(* CoDeSys 2.3.9.9 project: factory_a.pro *)
(* Libraries: standard.lib 4.10.05 11:14:46, Iecsfc.lib 13.4.06 15:51:28, Util.lib 1.6.07 09:40:58, SysLibTime.lib 18.7.05 09:39:56, SysTaskInfo.lib 18.7.05 09:39:56, SysLibMem.lib 18.7.05 09:39:56, SYSLIBCALLBACK.LIB 18.7.05 09:39:56, BusDiag.LIB 27.8.04 15:06:12, SysExt_AC500_V10.lib 1.7.05 16:17:10, SysInt_AC500_V10.LIB 2.6.06 10:49:48, Ethernet_AC500_V10.LIB 28.7.05 12:19:48 *)

(* PLC configuration (modules and I/O channels)
CPU parameters [AC500_CPU] node 0, in %IB0 out %QB0 {AutoRunType = On; ErrLEDType = On; CheckBatteryType = On; OutputsInStopType = Off in hardware and online; StopErrorClassType = No effect; WarmstartOnFK2Type = Off; FloatingPointExceptionType = E2 failure; IOSimulationModeType = Off; NumberRetainSegmentsType = 8; StartRetainM0Type = 0; EndRetainM0Type = 0; StartRetainM1Type = 0; EndRetainM1Type = 0; StartRetainM2Type = 0; EndRetainM2Type = 0; StartRetainM3Type = 0; EndRetainM3Type = 0; StartRetainM4Type = 0; EndRetainM4Type = 0; StartRetainM5Type = 0; EndRetainM5Type = 0; StartRetainM6Type = 0; EndRetainM6Type = 0; StartRetainM7Type = 0; EndRetainM7Type = 0}
AT %IW0 [WordInputNoSpace] Input 0-15
AT %IB0 [ByteInputNoSpace] Input 0-7
S0 AT %IX0.0 [BoolInput] Input 0
S1 AT %IX0.1 [BoolInput] Input 1
S2 AT %IX0.2 [BoolInput] Input 2
S3 AT %IX0.3 [BoolInput] Input 3
S4 AT %IX0.4 [BoolInput] Input 4
S5 AT %IX0.5 [BoolInput] Input 5
S6 AT %IX0.6 [BoolInput] Input 6
S7 AT %IX0.7 [BoolInput] Input 7
AT %IB1 [ByteInputNoSpace] Input 8-15
S8 AT %IX1.0 [BoolInput] Input 8
S9 AT %IX1.1 [BoolInput] Input 9
S10 AT %IX1.2 [BoolInput] Input 10
S11 AT %IX1.3 [BoolInput] Input 11
S12 AT %IX1.4 [BoolInput] Input 12
S13 AT %IX1.5 [BoolInput] Input 13
S14 AT %IX1.6 [BoolInput] Input 14
S15 AT %IX1.7 [BoolInput] Input 15
AT %IW1 [WordInputNoSpace] Input 16-31
AT %IB2 [ByteInputNoSpace] Input 16-23
AT %IX2.0 [BoolInput] Input 16
AT %IX2.1 [BoolInput] Input 17
AT %IX2.2 [BoolInput] Input 18
AT %IX2.3 [BoolInput] Input 19
AT %IX2.4 [BoolInput] Input 20
AT %IX2.5 [BoolInput] Input 21
AT %IX2.6 [BoolInput] Input 22
AT %IX2.7 [BoolInput] Input 23
AT %IB3 [ByteInputNoSpace] Input 24-31
AT %IX3.0 [BoolInput] Input 24
AT %IX3.1 [BoolInput] Input 25
AT %IX3.2 [BoolInput] Input 26
AT %IX3.3 [BoolInput] Input 27
AT %IX3.4 [BoolInput] Input 28
AT %IX3.5 [BoolInput] Input 29
AT %IX3.6 [BoolInput] Input 30
AT %IX3.7 [BoolInput] Input 31
AT %QW0 [WordOutputNoSpace] Output 16-31
AT %QB0 [ByteOutputNoSpace] Output 16-23
E0 AT %QX0.0 [BoolOutput] Output 16
E1B AT %QX0.1 [BoolOutput] Output 17
E2B AT %QX0.2 [BoolOutput] Output 18
E3 AT %QX0.3 [BoolOutput] Output 19
E4B AT %QX0.4 [BoolOutput] Output 20
E5B AT %QX0.5 [BoolOutput] Output 21
E6B AT %QX0.6 [BoolOutput] Output 22
E7B AT %QX0.7 [BoolOutput] Output 23
AT %QB1 [ByteOutputNoSpace] Output 24-31
AT %QX1.0 [BoolOutput] Output 24
E1F AT %QX1.1 [BoolOutput] Output 25
E2F AT %QX1.2 [BoolOutput] Output 26
AT %QX1.3 [BoolOutput] Output 27
E4F AT %QX1.4 [BoolOutput] Output 28
E5F AT %QX1.5 [BoolOutput] Output 29
E6F AT %QX1.6 [BoolOutput] Output 30
E7F AT %QX1.7 [BoolOutput] Output 31
AT %ID1 [DWordInput] Istwert/Actual value 1
AT %ID2 [DWordInput] Istwert/Actual value 2
AT %IB12 [ByteInputNoBits] Statusbyte/State byte 1
AT %IB13 [ByteInputNoBits] Statusbyte/State byte 2
AT %QD1 [DWordOutput] Startwert/Start value 1
AT %QD2 [DWordOutput] Endwert/End value 1
AT %QD3 [DWordOutput] Startwert/Start value 2
AT %QD4 [DWordOutput] Endwert/End value 2
AT %QB20 [ByteOutputNoBits] Steuerbyte/Control byte 1
AT %QB21 [ByteOutputNoBits] Steuerbyte/Control byte 2
AT %IW7 [WordInputNoSpace] Input 0-15
AT %IB14 [ByteInputNoSpace] Input 0-7
S16 AT %IX14.0 [BoolInput] Input 0
S17 AT %IX14.1 [BoolInput] Input 1
S18 AT %IX14.2 [BoolInput] Input 2
S19 AT %IX14.3 [BoolInput] Input 3
S20 AT %IX14.4 [BoolInput] Input 4
S21 AT %IX14.5 [BoolInput] Input 5
S22 AT %IX14.6 [BoolInput] Input 6
S23 AT %IX14.7 [BoolInput] Input 7
AT %IB15 [ByteInputNoSpace] Input 8-15
S24 AT %IX15.0 [BoolInput] Input 8
S25 AT %IX15.1 [BoolInput] Input 9
S26 AT %IX15.2 [BoolInput] Input 10
S27 AT %IX15.3 [BoolInput] Input 11
AT %IX15.4 [BoolInput] Input 12
AT %IX15.5 [BoolInput] Input 13
AT %IX15.6 [BoolInput] Input 14
SafetyLine_I215 AT %IX15.7 [BoolInput] Input 15
Digital In/Outputs - Inputs 16-31 [Module_16BitInput_16_31] node 1, in %IB16 out %QB22
  AT %IW8 [WordInputNoSpace] Input 16-31
  AT %IB16 [ByteInputNoSpace] Input 16-23
  AT %IX16.0 [BoolInput] Input 16
  AT %IX16.1 [BoolInput] Input 17
  AT %IX16.2 [BoolInput] Input 18
  AT %IX16.3 [BoolInput] Input 19
  AT %IX16.4 [BoolInput] Input 20
  AT %IX16.5 [BoolInput] Input 21
  AT %IX16.6 [BoolInput] Input 22
  AT %IX16.7 [BoolInput] Input 23
  AT %IB17 [ByteInputNoSpace] Input 24-31
  AT %IX17.0 [BoolInput] Input 24
  AT %IX17.1 [BoolInput] Input 25
  AT %IX17.2 [BoolInput] Input 26
  AT %IX17.3 [BoolInput] Input 27
  AT %IX17.4 [BoolInput] Input 28
  AT %IX17.5 [BoolInput] Input 29
  AT %IX17.6 [BoolInput] Input 30
  AT %IX17.7 [BoolInput] Input 31
AT %QW11 [WordOutputNoSpace] Output 16-31
AT %QB22 [ByteOutputNoSpace] Output 16-23
E8B AT %QX22.0 [BoolOutput] Output 16
E9U AT %QX22.1 [BoolOutput] Output 17
AT %QX22.2 [BoolOutput] Output 18
AT %QX22.3 [BoolOutput] Output 19
AT %QX22.4 [BoolOutput] Output 20
AT %QX22.5 [BoolOutput] Output 21
AT %QX22.6 [BoolOutput] Output 22
ALARM AT %QX22.7 [BoolOutput] Output 23
AT %QB23 [ByteOutputNoSpace] Output 24-31
E8F AT %QX23.0 [BoolOutput] Output 24
E9D AT %QX23.1 [BoolOutput] Output 25
AT %QX23.2 [BoolOutput] Output 26
AT %QX23.3 [BoolOutput] Output 27
AT %QX23.4 [BoolOutput] Output 28
AT %QX23.5 [BoolOutput] Output 29
AT %QX23.6 [BoolOutput] Output 30
AT %QX23.7 [BoolOutput] Output 31
AT %ID5 [DWordInput] Istwert/Actual value 1
AT %ID6 [DWordInput] Istwert/Actual value 2
AT %IB28 [ByteInputNoBits] Statusbyte/State byte 1
AT %IB29 [ByteInputNoBits] Statusbyte/State byte 2
AT %QD6 [DWordOutput] Startwert/Start value 1
AT %QD7 [DWordOutput] Endwert/End value 1
AT %QD8 [DWordOutput] Startwert/Start value 2
AT %QD9 [DWordOutput] Endwert/End value 2
AT %QB40 [ByteOutputNoBits] Steuerbyte/Control byte 1
AT %QB41 [ByteOutputNoBits] Steuerbyte/Control byte 2
COM1 - Online access [AC500_COM1_Programming] node 0, in %IB1000 out %QB1000 {COMEnableLoginType = Disabled; COMRTSctrlType = none; COMTLSType = 0; COMCDLYType = 0; COMCharTimeoutType = 0; COMTelEndSelType = none; COMTelEndValCharType = 16#00; COMTelEndValWertType = 0; COMChecksumType = none; COMHandshakeType = none; COMBaudType = 19200; COMParityType = none; COMDataBitType = 8; COMStopBitType = 1}
COM2 - Online access [AC500_COM2_Programming] node 1, in %IB2000 out %QB2000 {COMEnableLoginType = Disabled; COMRTSctrlType = none; COMTLSType = 0; COMCDLYType = 0; COMCharTimeoutType = 0; COMTelEndSelType = none; COMTelEndValCharType = 16#00; COMTelEndValWertType = 0; COMChecksumType = none; COMHandshakeType = none; COMBaudType = 19200; COMParityType = none; COMDataBitType = 8; COMStopBitType = 1}
FBP - none [AC500_FBP_None] node 2, in %IB3000 out %QB3000
MODBUS on TCP/IP [MODBUS_ETH_TCP] node 0, in %IB4000 out %QB4000 {ModbusCouplerOperatingModeType = Master/Slave; COMAdressType = 0; COMDisableWriteStartSeg0Type = 0; COMDisableWriteEndSeg0Type = 0; COMDisableReadStartSeg0Type = 0; COMDisableReadEndSeg0Type = 0; COMDisableWriteStartSeg1Type = 0; COMDisableWriteEndSeg1Type = 0; COMDisableReadStartSeg1Type = 0; COMDisableReadEndSeg1Type = 0}
External - none [AC500_Ext_Empty] node 1, in %IB4000 out %QB4000 {RunConfigFaultType = Yes; MaxWaitRunType = 3000; MinUpdateTimeType = 10; ReserveWord0Type = 0; ReserveWord1Type = 0; ReserveWord2Type = 0}
External - none [AC500_Ext_Empty] node 2, in %IB4000 out %QB4000 {RunConfigFaultType = Yes; MaxWaitRunType = 3000; MinUpdateTimeType = 10; ReserveWord0Type = 0; ReserveWord1Type = 0; ReserveWord2Type = 0}
*)

(* Global variable list: Global_Variables *)
VAR_GLOBAL

	(*Alarms*)
	PressFailureAlarm:BOOL;
	BASE_ALARM:BOOL := FALSE;
	DEFECT_ALARM:BOOL := FALSE;

	(*System variables*)
	AutomaticMode:BOOL :=TRUE;
	Emergency:BOOL :=FALSE;
	SFCInit: BOOL := FALSE;
	SFCReset: BOOL := FALSE;
	EffectorFailureTime: TIME := T#500ms;
	PressStarted:BOOL := FALSE;
	PressFailure:BOOL := FALSE;

	(*Variables for the automatic program*)
	START:BOOL :=FALSE;
	STOP:BOOL :=FALSE;
	RUN:BOOL :=FALSE;
	PRESS_READY:BOOL :=FALSE;
	DIAGNOSTICS_READY:BOOL :=FALSE;
	DEFECT_READY:BOOL :=FALSE;
	ELEVATOR_READY:BOOL :=FALSE;
	LOOK_FOR_PLATES:BOOL :=FALSE;
	NO_BASE_PLATES:BOOL :=FALSE;
	START_PRESS:BOOL :=FALSE;
	LOOK_FOR_BRICKS:BOOL :=FALSE;
	MISSING_BRICKS:BOOL :=FALSE;
	(* Faulty car flag (set by diagnostics) *)
	FAULTY_CAR:BOOL :=FALSE;
	(* Assembly line variables *)
	E0A:BOOL := FALSE;
	E0B:BOOL := FALSE;
	E0C:BOOL := FALSE;
	E0D:BOOL := FALSE;
	E0E:BOOL := FALSE;
	E0F:BOOL := FALSE;
	(* Safe motor variables*)
	E1FS:BOOL := FALSE;
	E1BS:BOOL := FALSE;
	E2FS:BOOL := FALSE;
	E2BS:BOOL := FALSE;
	E3S:BOOL := FALSE;
	E4FS:BOOL := FALSE;
	E4BS:BOOL := FALSE;
	E5FS:BOOL := FALSE;
	E5BS:BOOL := FALSE;
	E6FS:BOOL := FALSE;
	E6BS:BOOL := FALSE;
	E7FS:BOOL := FALSE;
	E7BS:BOOL := FALSE;
	E8FS:BOOL := FALSE;
	E8BS:BOOL := FALSE;
	E9US:BOOL := FALSE;
	E9DS:BOOL := FALSE;
	(* Car detection variables *)
	LOOK_FOR_CAR_PRESS:BOOL :=FALSE;
	CAR_DETECTED_PRESS:BOOL :=FALSE;
	CAR_ARRIVED_PRESS:BOOL :=FALSE;
	LOOK_FOR_CAR_DIAGNOSTICS:BOOL :=FALSE;
	CAR_ARRIVED_DIAGNOSTICS:BOOL :=FALSE;
	LOOK_FOR_CAR_DEFECT:BOOL :=FALSE;
	CAR_DETECTED_DEFECT:BOOL :=FALSE;
	CAR_ARRIVED_DEFECT:BOOL :=FALSE;
	LOOK_FOR_CAR_ELEVATOR:BOOL :=FALSE;
	CAR_DETECTED_ELEVATOR:BOOL :=FALSE;
	CAR_ARRIVED_ELEVATOR:BOOL :=FALSE;
END_VAR

(* POU PLC_PRG, LD *)
PROGRAM PLC_PRG
VAR
	automaticFalling: F_TRIG;
	automaticRising: R_TRIG;
	(* Tachometer *)
	Tacho: BOOL := TRUE;
	TachoTime: TIME := T#240ms;
	TachoTimer1: TON;
	TachoTimer2: TON;
	(* Effector Failure *)
	EffectorFailure: BOOL;
	E1FailureTimer1: TON;
	E1FailureTimer2: TON;
	E1Failure: BOOL;
	E2FailureTimer1: TON;
	E2FailureTimer2: TON;
	E2Failure: BOOL;
	E3FailureTimer: TON;
	E3Failure: BOOL;
	E4FailureTimer1: TON;
	E4FailureTimer2: TON;
	E4Failure: BOOL;
	E5FailureTimer1: TON;
	E5FailureTimer2: TON;
	E5Failure: BOOL;
	E6FailureTimer1: TON;
	E6FailureTimer2: TON;
	E6Failure: BOOL;
	E7FailureTimer1: TON;
	E7FailureTimer2: TON;
	E7Failure: BOOL;
	E8FailureTimer1: TON;
	E8FailureTimer2: TON;
	E8Failure: BOOL;
	E9FailureTimer1: TON;
	E9FailureTimer2: TON;
	E9Failure: BOOL;

	(*Safty press timer, The max press time when press is stuck*)
	(* MaxPressTime:TIME := T#700ms;

	SafetyPressTimer2: TON;
	SafetyPressTimer1: TON;
	Output1: BOOL; *)
END_VAR
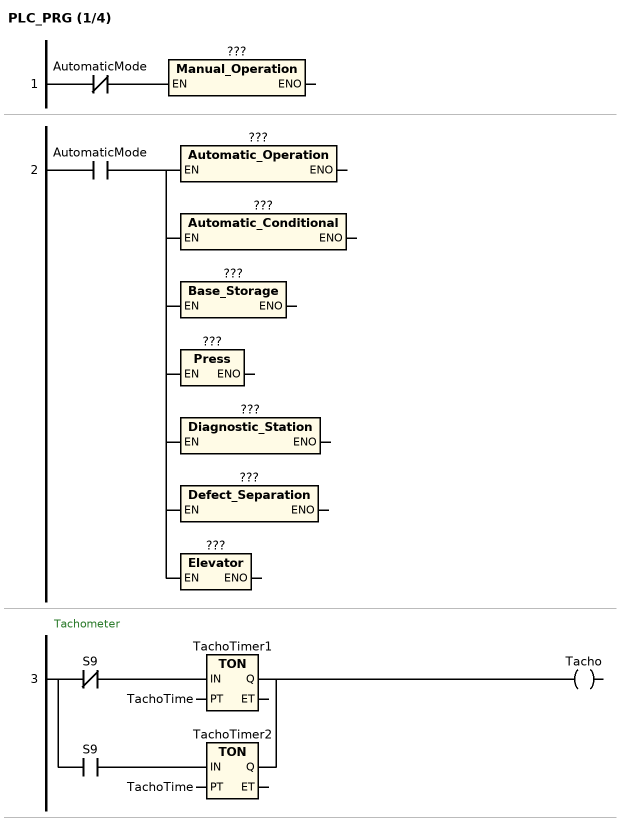
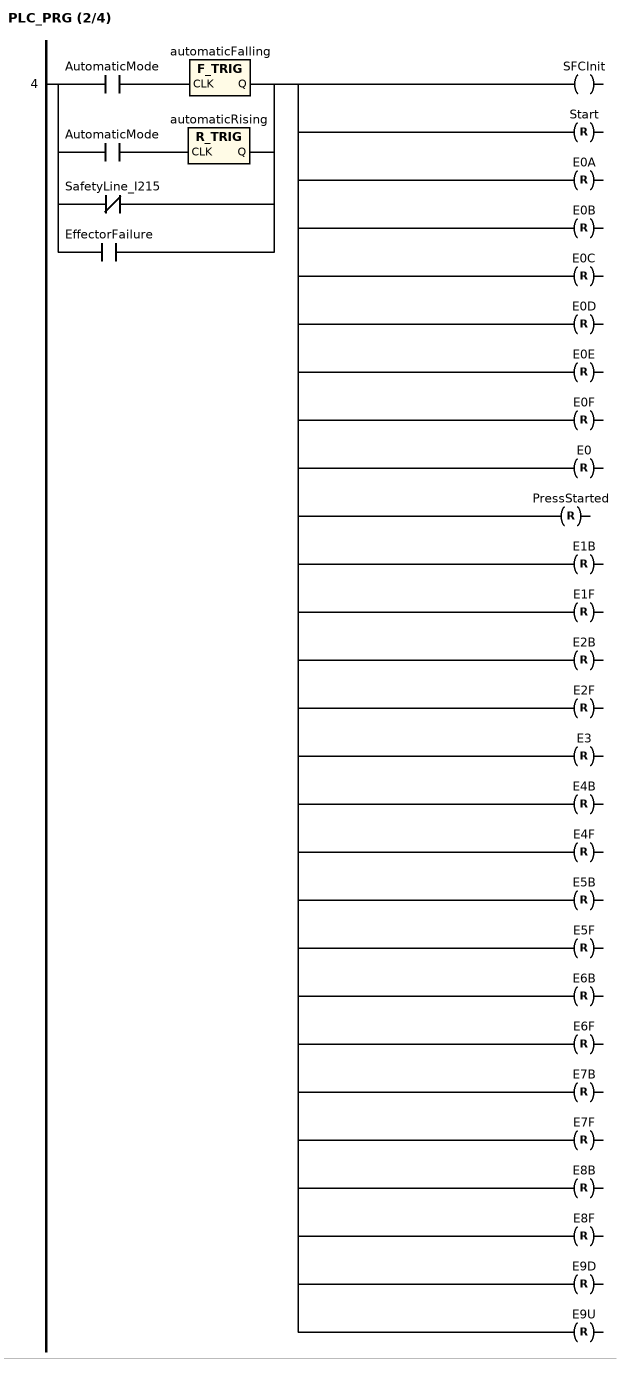
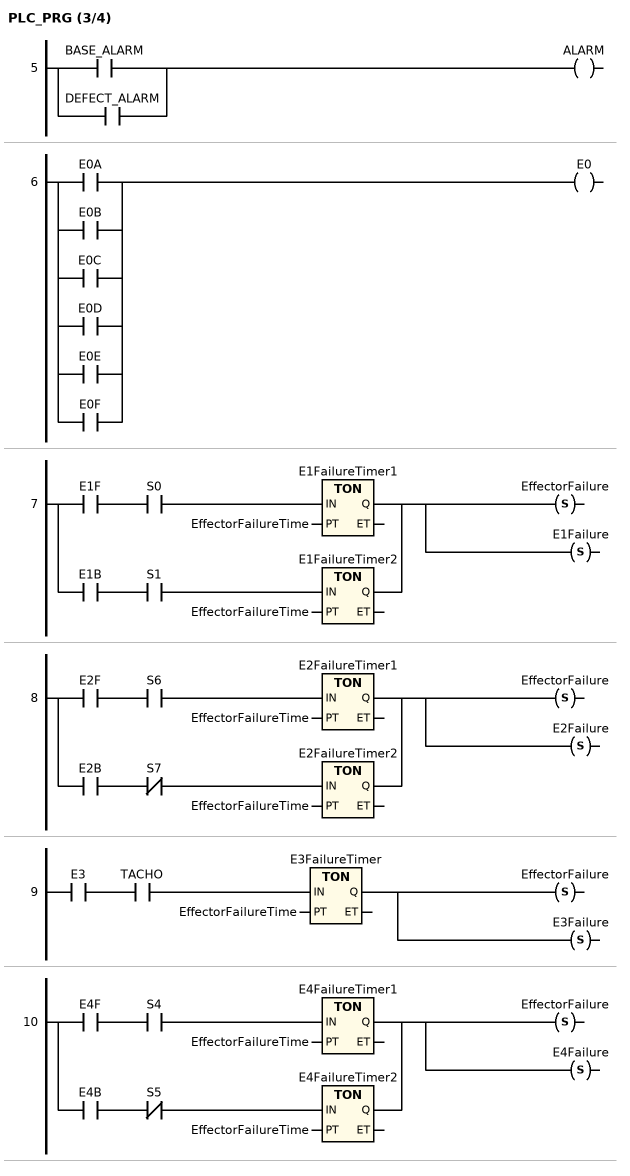
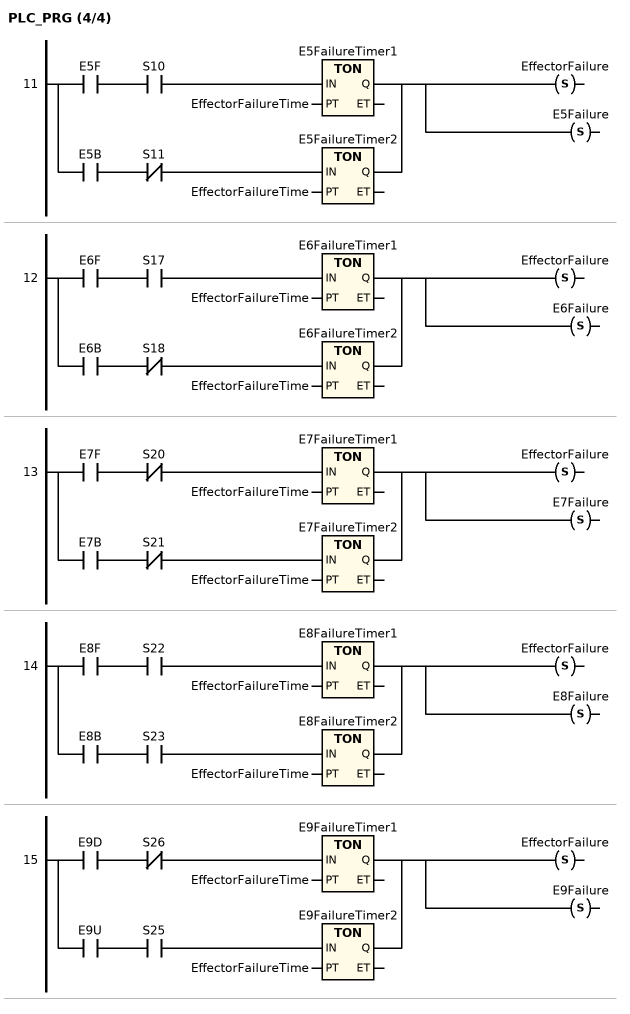
_LD_ (* Ladder Diagram *)
NETWORK 1
	[/AutomaticMode]
		EN --- ???:Manual_Operation()
NETWORK 2
	[AutomaticMode]
		EN --- ???:Automatic_Operation()
		EN --- ???:Automatic_Conditional()
		EN --- ???:Base_Storage()
		EN --- ???:Press()
		EN --- ???:Diagnostic_Station()
		EN --- ???:Defect_Separation()
		EN --- ???:Elevator()
NETWORK 3 (* Tachometer *)
	{ [/S9] - TachoTimer1:TON(IN: *, PT: TachoTime) | [S9] - TachoTimer2:TON(IN: *, PT: TachoTime) } --- (Tacho)
NETWORK 4
	{ [AutomaticMode] - automaticFalling:F_TRIG(CLK: *) | [AutomaticMode] - automaticRising:R_TRIG(CLK: *) | [/SafetyLine_I215] | [EffectorFailure] } --- (SFCInit) (R Start) (R E0A) (R E0B) (R E0C) (R E0D) (R E0E) (R E0F) (R E0) (R PressStarted) (R E1B) (R E1F) (R E2B) (R E2F) (R E3) (R E4B) (R E4F) (R E5B) (R E5F) (R E6B) (R E6F) (R E7B) (R E7F) (R E8B) (R E8F) (R E9D) (R E9U)
NETWORK 5
	{ [BASE_ALARM] | [DEFECT_ALARM] } --- (ALARM)
NETWORK 6
	{ [E0A] | [E0B] | [E0C] | [E0D] | [E0E] | [E0F] } --- (E0)
NETWORK 7
	{ [E1F] - [S0] - E1FailureTimer1:TON(IN: *, PT: EffectorFailureTime) | [E1B] - [S1] - E1FailureTimer2:TON(IN: *, PT: EffectorFailureTime) } --- (S EffectorFailure) (S E1Failure)
NETWORK 8
	{ [E2F] - [S6] - E2FailureTimer1:TON(IN: *, PT: EffectorFailureTime) | [E2B] - [/S7] - E2FailureTimer2:TON(IN: *, PT: EffectorFailureTime) } --- (S EffectorFailure) (S E2Failure)
NETWORK 9
	[E3] - [TACHO] - E3FailureTimer:TON(IN: *, PT: EffectorFailureTime) --- (S EffectorFailure) (S E3Failure)
NETWORK 10
	{ [E4F] - [S4] - E4FailureTimer1:TON(IN: *, PT: EffectorFailureTime) | [E4B] - [/S5] - E4FailureTimer2:TON(IN: *, PT: EffectorFailureTime) } --- (S EffectorFailure) (S E4Failure)
NETWORK 11
	{ [E5F] - [S10] - E5FailureTimer1:TON(IN: *, PT: EffectorFailureTime) | [E5B] - [/S11] - E5FailureTimer2:TON(IN: *, PT: EffectorFailureTime) } --- (S EffectorFailure) (S E5Failure)
NETWORK 12
	{ [E6F] - [S17] - E6FailureTimer1:TON(IN: *, PT: EffectorFailureTime) | [E6B] - [/S18] - E6FailureTimer2:TON(IN: *, PT: EffectorFailureTime) } --- (S EffectorFailure) (S E6Failure)
NETWORK 13
	{ [E7F] - [/S20] - E7FailureTimer1:TON(IN: *, PT: EffectorFailureTime) | [E7B] - [/S21] - E7FailureTimer2:TON(IN: *, PT: EffectorFailureTime) } --- (S EffectorFailure) (S E7Failure)
NETWORK 14
	{ [E8F] - [S22] - E8FailureTimer1:TON(IN: *, PT: EffectorFailureTime) | [E8B] - [S23] - E8FailureTimer2:TON(IN: *, PT: EffectorFailureTime) } --- (S EffectorFailure) (S E8Failure)
NETWORK 15
	{ [E9D] - [/S26] - E9FailureTimer1:TON(IN: *, PT: EffectorFailureTime) | [E9U] - [S25] - E9FailureTimer2:TON(IN: *, PT: EffectorFailureTime) } --- (S EffectorFailure) (S E9Failure)
_END_LD_
(* the same logic as Structured Text *)
(* Network 1: see the listing above *)
(* Network 2: see the listing above *)
(* Network 3 *)
TachoTimer1(IN := NOT S9, PT := TachoTime);
TachoTimer2(IN := S9, PT := TachoTime);
Tacho := TachoTimer1.Q OR TachoTimer2.Q;
(* Network 4 *)
automaticFalling(CLK := AutomaticMode);
automaticRising(CLK := AutomaticMode);
SFCInit := automaticFalling.Q OR automaticRising.Q OR NOT SafetyLine_I215 OR EffectorFailure;
IF SFCInit THEN Start := FALSE; E0A := FALSE; E0B := FALSE; E0C := FALSE; E0D := FALSE; E0E := FALSE; E0F := FALSE; E0 := FALSE; PressStarted := FALSE; E1B := FALSE; E1F := FALSE; E2B := FALSE; E2F := FALSE; E3 := FALSE; E4B := FALSE; E4F := FALSE; E5B := FALSE; E5F := FALSE; E6B := FALSE; E6F := FALSE; E7B := FALSE; E7F := FALSE; E8B := FALSE; E8F := FALSE; E9D := FALSE; E9U := FALSE; END_IF;
(* Network 5 *)
ALARM := BASE_ALARM OR DEFECT_ALARM;
(* Network 6 *)
E0 := E0A OR E0B OR E0C OR E0D OR E0E OR E0F;
(* Network 7 *)
E1FailureTimer1(IN := E1F AND S0, PT := EffectorFailureTime);
E1FailureTimer2(IN := E1B AND S1, PT := EffectorFailureTime);
IF E1FailureTimer1.Q OR E1FailureTimer2.Q THEN EffectorFailure := TRUE; E1Failure := TRUE; END_IF;
(* Network 8 *)
E2FailureTimer1(IN := E2F AND S6, PT := EffectorFailureTime);
E2FailureTimer2(IN := E2B AND NOT S7, PT := EffectorFailureTime);
IF E2FailureTimer1.Q OR E2FailureTimer2.Q THEN EffectorFailure := TRUE; E2Failure := TRUE; END_IF;
(* Network 9 *)
E3FailureTimer(IN := E3 AND TACHO, PT := EffectorFailureTime);
IF E3FailureTimer.Q THEN EffectorFailure := TRUE; E3Failure := TRUE; END_IF;
(* Network 10 *)
E4FailureTimer1(IN := E4F AND S4, PT := EffectorFailureTime);
E4FailureTimer2(IN := E4B AND NOT S5, PT := EffectorFailureTime);
IF E4FailureTimer1.Q OR E4FailureTimer2.Q THEN EffectorFailure := TRUE; E4Failure := TRUE; END_IF;
(* Network 11 *)
E5FailureTimer1(IN := E5F AND S10, PT := EffectorFailureTime);
E5FailureTimer2(IN := E5B AND NOT S11, PT := EffectorFailureTime);
IF E5FailureTimer1.Q OR E5FailureTimer2.Q THEN EffectorFailure := TRUE; E5Failure := TRUE; END_IF;
(* Network 12 *)
E6FailureTimer1(IN := E6F AND S17, PT := EffectorFailureTime);
E6FailureTimer2(IN := E6B AND NOT S18, PT := EffectorFailureTime);
IF E6FailureTimer1.Q OR E6FailureTimer2.Q THEN EffectorFailure := TRUE; E6Failure := TRUE; END_IF;
(* Network 13 *)
E7FailureTimer1(IN := E7F AND NOT S20, PT := EffectorFailureTime);
E7FailureTimer2(IN := E7B AND NOT S21, PT := EffectorFailureTime);
IF E7FailureTimer1.Q OR E7FailureTimer2.Q THEN EffectorFailure := TRUE; E7Failure := TRUE; END_IF;
(* Network 14 *)
E8FailureTimer1(IN := E8F AND S22, PT := EffectorFailureTime);
E8FailureTimer2(IN := E8B AND S23, PT := EffectorFailureTime);
IF E8FailureTimer1.Q OR E8FailureTimer2.Q THEN EffectorFailure := TRUE; E8Failure := TRUE; END_IF;
(* Network 15 *)
E9FailureTimer1(IN := E9D AND NOT S26, PT := EffectorFailureTime);
E9FailureTimer2(IN := E9U AND S25, PT := EffectorFailureTime);
IF E9FailureTimer1.Q OR E9FailureTimer2.Q THEN EffectorFailure := TRUE; E9Failure := TRUE; END_IF;
END_PROGRAM

(* POU Manual_Operation, SFC *)
PROGRAM Manual_Operation
VAR
	StorageAlarmTime:TIME :=T#2S;
	(*E0: Assembly line*)
	(*Not in SFC.Using  E0A directly*)
	(*E1: Base pusher*)
	buttonE1Fwd: BOOL := FALSE;
	buttonE1Bwd: BOOL := FALSE;
	(*E2: Undercarriage pusher*)
	buttonE2Fwd: BOOL := FALSE;
	buttonE2Bwd: BOOL := FALSE;
	(*E3: Press
	Observe! that S8 is active low*)
	buttonE3Press: BOOL := FALSE;
	(*E4: Press pusher*)
	buttonE4Fwd: BOOL := FALSE;
	buttonE4Bwd: BOOL := FALSE;
	(*E5: Press bar*)
	buttonE5Fwd: BOOL := FALSE;
	buttonE5Bwd: BOOL := FALSE;
	(*E6: Diagnostic bar
	Observe! that InEngine6 has NOT inverted contact*)
	buttonE6Fwd: BOOL := FALSE;
	buttonE6Bwd: BOOL := FALSE;
	(*E7: Defect pusher*)
	TimeOutStorage: BOOL := FALSE;
	buttonE7Fwd: BOOL := FALSE;
	buttonE7Bwd: BOOL := FALSE;
	(*E8: Defect bar*)
	buttonE8Fwd: BOOL := FALSE;
	buttonE8Bwd: BOOL := FALSE;
	(*E9: Elevator*)
	buttonE9Up: BOOL := FALSE;
	buttonE9Down: BOOL := FALSE;
END_VAR
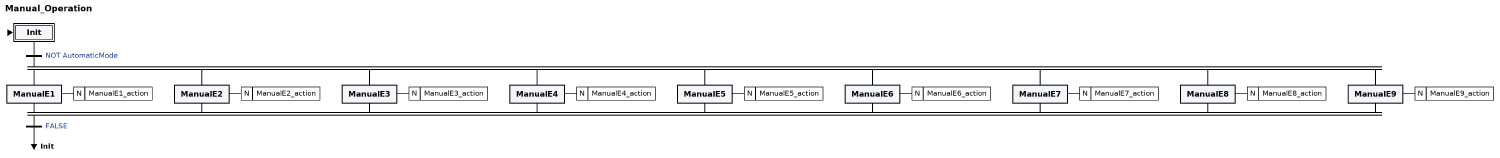
INITIAL_STEP Init:
END_STEP
TRANSITION FROM Init TO (ManualE1, ManualE2, ManualE3, ManualE4, ManualE5, ManualE6, ManualE7, ManualE8, ManualE9) := NOT AutomaticMode;
END_TRANSITION
STEP ManualE1:
	ManualE1_action(N);
END_STEP
STEP ManualE2:
	ManualE2_action(N);
END_STEP
STEP ManualE3:
	ManualE3_action(N);
END_STEP
STEP ManualE4:
	ManualE4_action(N);
END_STEP
STEP ManualE5:
	ManualE5_action(N);
END_STEP
STEP ManualE6:
	ManualE6_action(N);
END_STEP
STEP ManualE7:
	ManualE7_action(N);
END_STEP
STEP ManualE8:
	ManualE8_action(N);
END_STEP
STEP ManualE9:
	ManualE9_action(N);
END_STEP
TRANSITION FROM (ManualE1, ManualE2, ManualE3, ManualE4, ManualE5, ManualE6, ManualE7, ManualE8, ManualE9) TO Init := FALSE;
END_TRANSITION

ACTION ManualE1_action:
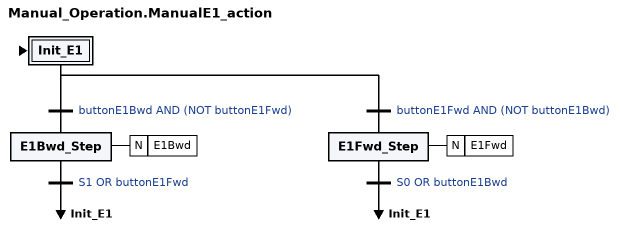
INITIAL_STEP Init_E1:
END_STEP
TRANSITION FROM Init_E1 TO E1Bwd_Step := buttonE1Bwd AND (NOT buttonE1Fwd);
END_TRANSITION
TRANSITION FROM Init_E1 TO E1Fwd_Step := buttonE1Fwd AND (NOT buttonE1Bwd);
END_TRANSITION
STEP E1Bwd_Step:
	E1Bwd(N);
END_STEP
TRANSITION FROM E1Bwd_Step TO Init_E1 := S1 OR buttonE1Fwd;
END_TRANSITION
STEP E1Fwd_Step:
	E1Fwd(N);
END_STEP
TRANSITION FROM E1Fwd_Step TO Init_E1 := S0 OR buttonE1Bwd;
END_TRANSITION
END_ACTION

ACTION ManualE2_action:
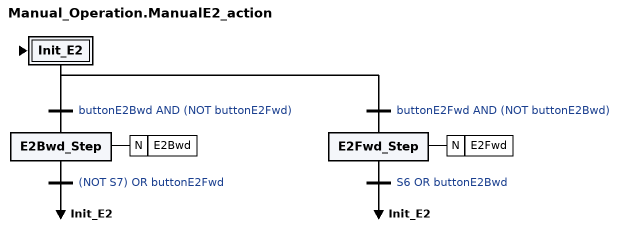
INITIAL_STEP Init_E2:
END_STEP
TRANSITION FROM Init_E2 TO E2Bwd_Step := buttonE2Bwd AND (NOT buttonE2Fwd);
END_TRANSITION
TRANSITION FROM Init_E2 TO E2Fwd_Step := buttonE2Fwd AND (NOT buttonE2Bwd);
END_TRANSITION
STEP E2Bwd_Step:
	E2Bwd(N);
END_STEP
TRANSITION FROM E2Bwd_Step TO Init_E2 := (NOT S7) OR buttonE2Fwd;
END_TRANSITION
STEP E2Fwd_Step:
	E2Fwd(N);
END_STEP
TRANSITION FROM E2Fwd_Step TO Init_E2 := S6 OR buttonE2Bwd;
END_TRANSITION
END_ACTION

ACTION ManualE3_action:
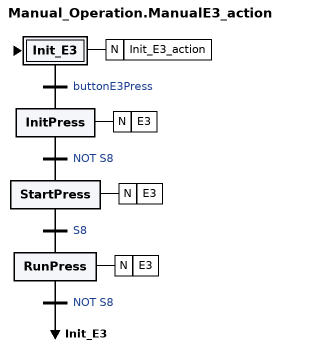
INITIAL_STEP Init_E3:
	Init_E3_action(N);
END_STEP
TRANSITION FROM Init_E3 TO InitPress := buttonE3Press;
END_TRANSITION
STEP InitPress:
	E3(N);
END_STEP
TRANSITION FROM InitPress TO StartPress := NOT S8;
END_TRANSITION
STEP StartPress:
	E3(N);
END_STEP
TRANSITION FROM StartPress TO RunPress := S8;
END_TRANSITION
STEP RunPress:
	E3(N);
END_STEP
TRANSITION FROM RunPress TO Init_E3 := NOT S8;
END_TRANSITION

ACTION Init_E3_action:
PressFailure :=FALSE;
END_ACTION
END_ACTION

ACTION ManualE4_action:
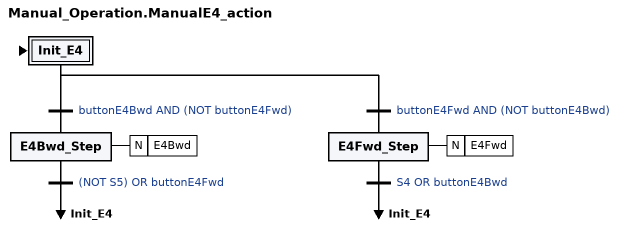
INITIAL_STEP Init_E4:
END_STEP
TRANSITION FROM Init_E4 TO E4Bwd_Step := buttonE4Bwd AND (NOT buttonE4Fwd);
END_TRANSITION
TRANSITION FROM Init_E4 TO E4Fwd_Step := buttonE4Fwd AND (NOT buttonE4Bwd);
END_TRANSITION
STEP E4Bwd_Step:
	E4Bwd(N);
END_STEP
TRANSITION FROM E4Bwd_Step TO Init_E4 := (NOT S5) OR buttonE4Fwd;
END_TRANSITION
STEP E4Fwd_Step:
	E4Fwd(N);
END_STEP
TRANSITION FROM E4Fwd_Step TO Init_E4 := S4 OR buttonE4Bwd;
END_TRANSITION
END_ACTION

ACTION ManualE5_action:
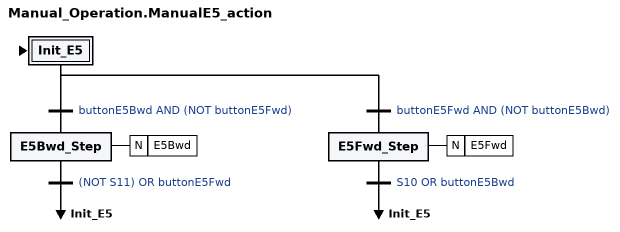
INITIAL_STEP Init_E5:
END_STEP
TRANSITION FROM Init_E5 TO E5Bwd_Step := buttonE5Bwd AND (NOT buttonE5Fwd);
END_TRANSITION
TRANSITION FROM Init_E5 TO E5Fwd_Step := buttonE5Fwd AND (NOT buttonE5Bwd);
END_TRANSITION
STEP E5Bwd_Step:
	E5Bwd(N);
END_STEP
TRANSITION FROM E5Bwd_Step TO Init_E5 := (NOT S11) OR buttonE5Fwd;
END_TRANSITION
STEP E5Fwd_Step:
	E5Fwd(N);
END_STEP
TRANSITION FROM E5Fwd_Step TO Init_E5 := S10 OR buttonE5Bwd;
END_TRANSITION
END_ACTION

ACTION ManualE6_action:
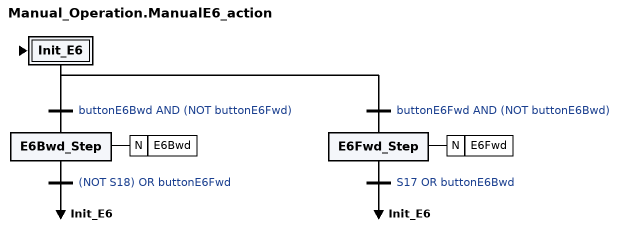
INITIAL_STEP Init_E6:
END_STEP
TRANSITION FROM Init_E6 TO E6Bwd_Step := buttonE6Bwd AND (NOT buttonE6Fwd);
END_TRANSITION
TRANSITION FROM Init_E6 TO E6Fwd_Step := buttonE6Fwd AND (NOT buttonE6Bwd);
END_TRANSITION
STEP E6Bwd_Step:
	E6Bwd(N);
END_STEP
TRANSITION FROM E6Bwd_Step TO Init_E6 := (NOT S18) OR buttonE6Fwd;
END_TRANSITION
STEP E6Fwd_Step:
	E6Fwd(N);
END_STEP
TRANSITION FROM E6Fwd_Step TO Init_E6 := S17 OR buttonE6Bwd;
END_TRANSITION
END_ACTION

ACTION ManualE7_action:
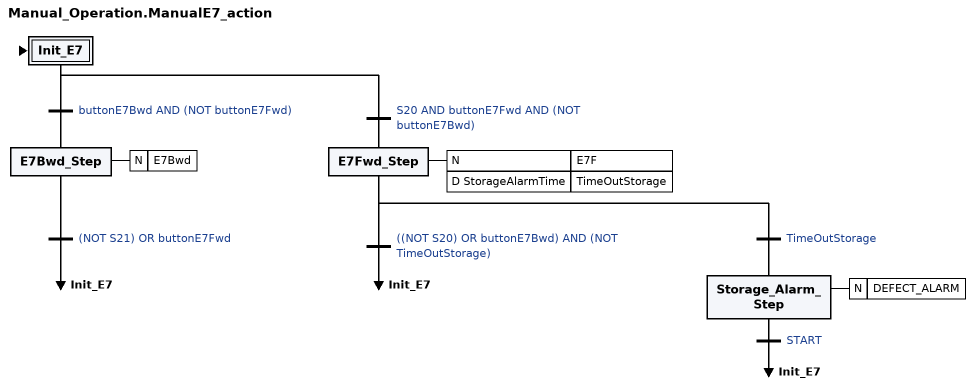
INITIAL_STEP Init_E7:
END_STEP
TRANSITION FROM Init_E7 TO E7Bwd_Step := buttonE7Bwd AND (NOT buttonE7Fwd);
END_TRANSITION
TRANSITION FROM Init_E7 TO E7Fwd_Step := S20 AND buttonE7Fwd AND (NOT buttonE7Bwd);
END_TRANSITION
STEP E7Bwd_Step:
	E7Bwd(N);
END_STEP
TRANSITION FROM E7Bwd_Step TO Init_E7 := (NOT S21) OR buttonE7Fwd;
END_TRANSITION
STEP E7Fwd_Step:
	E7F(N);
	TimeOutStorage(D, StorageAlarmTime);
END_STEP
TRANSITION FROM E7Fwd_Step TO Init_E7 := ((NOT S20) OR buttonE7Bwd) AND (NOT TimeOutStorage);
END_TRANSITION
TRANSITION FROM E7Fwd_Step TO Storage_Alarm_Step := TimeOutStorage;
END_TRANSITION
STEP Storage_Alarm_Step:
	DEFECT_ALARM(N);
END_STEP
TRANSITION FROM Storage_Alarm_Step TO Init_E7 := START;
END_TRANSITION
END_ACTION

ACTION ManualE8_action:
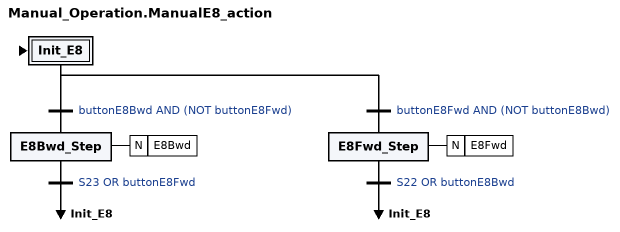
INITIAL_STEP Init_E8:
END_STEP
TRANSITION FROM Init_E8 TO E8Bwd_Step := buttonE8Bwd AND (NOT buttonE8Fwd);
END_TRANSITION
TRANSITION FROM Init_E8 TO E8Fwd_Step := buttonE8Fwd AND (NOT buttonE8Bwd);
END_TRANSITION
STEP E8Bwd_Step:
	E8Bwd(N);
END_STEP
TRANSITION FROM E8Bwd_Step TO Init_E8 := S23 OR buttonE8Fwd;
END_TRANSITION
STEP E8Fwd_Step:
	E8Fwd(N);
END_STEP
TRANSITION FROM E8Fwd_Step TO Init_E8 := S22 OR buttonE8Bwd;
END_TRANSITION
END_ACTION

ACTION ManualE9_action:
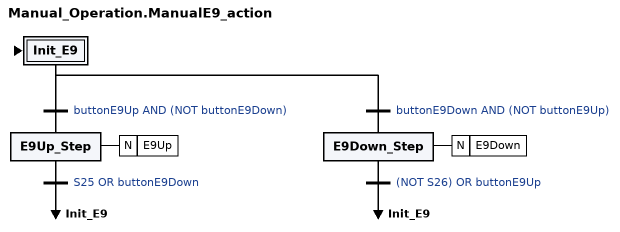
INITIAL_STEP Init_E9:
END_STEP
TRANSITION FROM Init_E9 TO E9Up_Step := buttonE9Up AND (NOT buttonE9Down);
END_TRANSITION
TRANSITION FROM Init_E9 TO E9Down_Step := buttonE9Down AND (NOT buttonE9Up);
END_TRANSITION
STEP E9Up_Step:
	E9Up(N);
END_STEP
TRANSITION FROM E9Up_Step TO Init_E9 := S25 OR buttonE9Down;
END_TRANSITION
STEP E9Down_Step:
	E9Down(N);
END_STEP
TRANSITION FROM E9Down_Step TO Init_E9 := (NOT S26) OR buttonE9Up;
END_TRANSITION
END_ACTION
END_PROGRAM
ACTION E1Bwd:
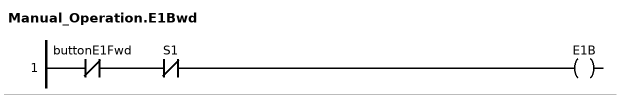
_LD_ (* Ladder Diagram *)
NETWORK 1
	[/buttonE1Fwd] - [/S1] --- (E1B)
_END_LD_
(* the same logic as Structured Text *)
(* Network 1 *)
E1B := NOT buttonE1Fwd AND NOT S1;
END_ACTION
ACTION E1Fwd:
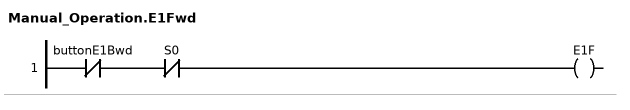
_LD_ (* Ladder Diagram *)
NETWORK 1
	[/buttonE1Bwd] - [/S0] --- (E1F)
_END_LD_
(* the same logic as Structured Text *)
(* Network 1 *)
E1F := NOT buttonE1Bwd AND NOT S0;
END_ACTION
ACTION E2Bwd:
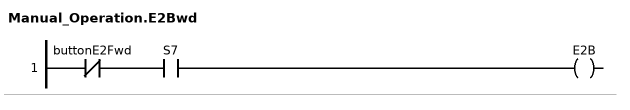
_LD_ (* Ladder Diagram *)
NETWORK 1
	[/buttonE2Fwd] - [S7] --- (E2B)
_END_LD_
(* the same logic as Structured Text *)
(* Network 1 *)
E2B := NOT buttonE2Fwd AND S7;
END_ACTION
ACTION E2Fwd:
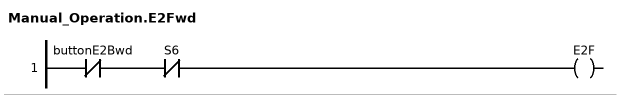
_LD_ (* Ladder Diagram *)
NETWORK 1
	[/buttonE2Bwd] - [/S6] --- (E2F)
_END_LD_
(* the same logic as Structured Text *)
(* Network 1 *)
E2F := NOT buttonE2Bwd AND NOT S6;
END_ACTION
ACTION E4Bwd:
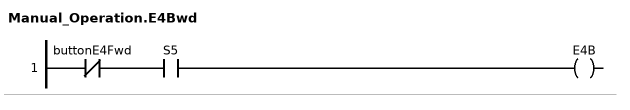
_LD_ (* Ladder Diagram *)
NETWORK 1
	[/buttonE4Fwd] - [S5] --- (E4B)
_END_LD_
(* the same logic as Structured Text *)
(* Network 1 *)
E4B := NOT buttonE4Fwd AND S5;
END_ACTION
ACTION E4Fwd:
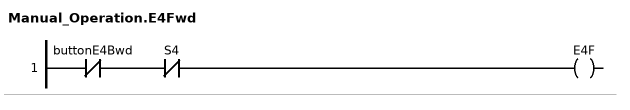
_LD_ (* Ladder Diagram *)
NETWORK 1
	[/buttonE4Bwd] - [/S4] --- (E4F)
_END_LD_
(* the same logic as Structured Text *)
(* Network 1 *)
E4F := NOT buttonE4Bwd AND NOT S4;
END_ACTION
ACTION E5Bwd:
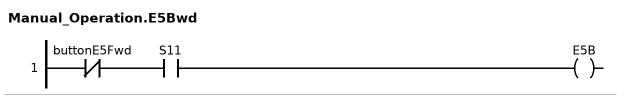
_LD_ (* Ladder Diagram *)
NETWORK 1
	[/buttonE5Fwd] - [S11] --- (E5B)
_END_LD_
(* the same logic as Structured Text *)
(* Network 1 *)
E5B := NOT buttonE5Fwd AND S11;
END_ACTION
ACTION E5Fwd:
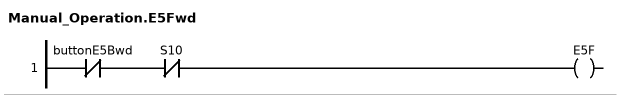
_LD_ (* Ladder Diagram *)
NETWORK 1
	[/buttonE5Bwd] - [/S10] --- (E5F)
_END_LD_
(* the same logic as Structured Text *)
(* Network 1 *)
E5F := NOT buttonE5Bwd AND NOT S10;
END_ACTION
ACTION E6Bwd:
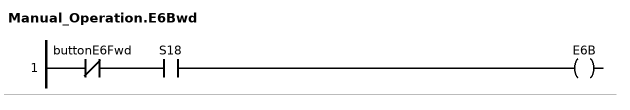
_LD_ (* Ladder Diagram *)
NETWORK 1
	[/buttonE6Fwd] - [S18] --- (E6B)
_END_LD_
(* the same logic as Structured Text *)
(* Network 1 *)
E6B := NOT buttonE6Fwd AND S18;
END_ACTION
ACTION E6Fwd:
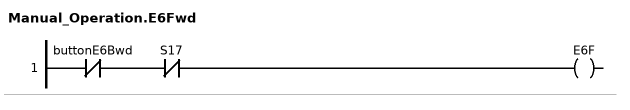
_LD_ (* Ladder Diagram *)
NETWORK 1
	[/buttonE6Bwd] - [/S17] --- (E6F)
_END_LD_
(* the same logic as Structured Text *)
(* Network 1 *)
E6F := NOT buttonE6Bwd AND NOT S17;
END_ACTION
ACTION E7Bwd:
